TYPE ST_MainCharmber :
STRUCT
END_STRUCT
END_TYPE

(* stored: Version 1.1.0.1, ProductVersion 3.1.4024.12
   DUT ST_MainCharmber: Id {480b7c1f-b7f8-4cac-87b5-297075ab26ac} *)
